(* PLC project EPEC_CU1.project, CODESYS V3.5 SP10, author XXXX *)
(* stored: creationDateTime 2025-02-24T16:09:32.0642752-06:00, modificationDateTime 2025-02-24T16:09:32.0642752-06:00, organization XXXX *)

TYPE FastParameters : STRUCT
  FastParameter1 : BYTE;
  FastParameter2 : WORD;
  FastParameter3 : DWORD;
END_STRUCT;
END_TYPE

(* This PRG contains non safety-related code. The following attribute is autogenerated. Do not remove. *)
{attribute 'location' := '16#800'}
PROGRAM Main

                    
(*
EC44 REF and output group are application controlled using product specific HW diagnostic program.
Following example can be used for controlling. Add application specific conditions.

EPEC_SHWD.S_EC44_Diagnostic.i_OutputGroup1Control := G_StatusFlags.SystemOk;
EPEC_SHWD.S_EC44_Diagnostic.i_RefVoltageControl := G_StatusFlags.SystemOk;

For more information, see Epec programming manual's How to guides.
*)										
										
                  
END_PROGRAM

(* This PRG contains non safety-related code. The following attribute is autogenerated. Do not remove. *)
{attribute 'location' := '16#800'}
PROGRAM MainInit
  VAR_OUTPUT
    o_MainInitReady : BOOL := FALSE;
  END_VAR

                    o_MainInitReady := TRUE;
                  
END_PROGRAM

(* NOTE! NOTE! NOTE! NOTE! NOTE! NOTE! NOTE! NOTE! NOTE! NOTE! NOTE! This object is created by Epec MultiTool User changes are overwritten when project is imported Content: - Input pin data update. This PRG contains non safety-related code. The following attribute is autogenerated. Do not remove. *)
{attribute 'hide_all_locals'}
{attribute 'location' := '16#800'}
PROGRAM Inputs
  VAR_INPUT
    i_Enable : BOOL := TRUE;
    i_Initialize : BOOL := TRUE;
  END_VAR
  VAR_OUTPUT
    o_InitReady : BOOL := FALSE;
    o_AI_POWER1_SUPPLY_Diagnostic : DWORD;  (* Measurent for power switch input voltage [unscaled] *)
    o_AI_POWER1_OUTPUT_Diagnostic : DWORD;  (* Measurement for power switch output voltage [unscaled]. *)
    o_AI_REF_OUTPUT_MAIN_Diagnostic : DWORD;  (* Measurement for selectable reference voltage (5/10V) [unscaled]. *)
    o_TEMP_PCB_MAIN_Diagnostic : DWORD;  (* Measurement for PCB temperature 1 [unscaled] *)
    o_TEMP_PCB_RED_Diagnostic : DWORD;  (* Measurement for PCB temperature 2 [unscaled] *)
    o_VIN_1_1_Diagnostic : DWORD;  (* Measurement for supply pin voltage [unscaled] *)
    o_VIN_POWER_Diagnostic : DWORD;  (* Measurement for Vin power [unscaled] *)
    o_TEMP_MCU_Diagnostic : DINT;  (* Measurement for MCU temperature [0.1C] *)
    o_AI_5VAN_Diagnostic : DWORD;  (* Measurement for 5VAN voltage [unscaled] *)
    o_AI_SBC_TEMP_Diagnostic : DINT;  (* SBC temperature [0.1 C] *)
  END_VAR
  VAR
    AI_POWER1_SUPPLY_Diagnostic : DWORD;  (* Measurent for power switch input voltage (Mapped variable) *)
    AI_POWER1_OUTPUT_Diagnostic : DWORD;  (* Measurement for power switch output voltage (Mapped variable).. *)
    AI_REF_OUTPUT_MAIN_Diagnostic : DWORD;  (* Measurement for selectable reference voltage (5/10V). (Mapped variable) *)
    TEMP_PCB_MAIN_Diagnostic : DWORD;  (* Measurement for PCB temperature 1 (Mapped variable) *)
    TEMP_PCB_RED_Diagnostic : DWORD;  (* Measurement for PCB temperature 2 (Mapped variable) *)
    VIN_1_1_Diagnostic : DWORD;  (* Measurement for supply pin voltage (Mapped variable) *)
    VIN_POWER_Diagnostic : DWORD;  (* Measurement for Vin power (Mapped variable) *)
    TEMP_MCU_Diagnostic : DINT;  (* Measurement for MCU temperature (Mapped variable) *)
    AI_5VAN_Diagnostic : DWORD;  (* Measurement for 5VAN voltage (Mapped variable) *)
    AI_SBC_TEMP_Diagnostic : DINT;  (* SBC temperature [0.1 C] *)
  END_VAR

                    IF(i_Initialize) THEN
	o_InitReady:= TRUE;
¤#INIT_INPUTS_INIT#¤  
ELSE
¤#INIT_INPUTS_CODE#¤  
END_IF

                  
END_PROGRAM

CONFIGURATION Device
  RESOURCE Application ON PLC
    TASK NonSafePRG_TASK(INTERVAL := T#10ms, PRIORITY := 1);
    PROGRAM PLC_PRG WITH NonSafePRG_TASK : PLC_PRG;
  END_RESOURCE
END_CONFIGURATION
